Universal Robots PolyScope program: Bridge_big.urp

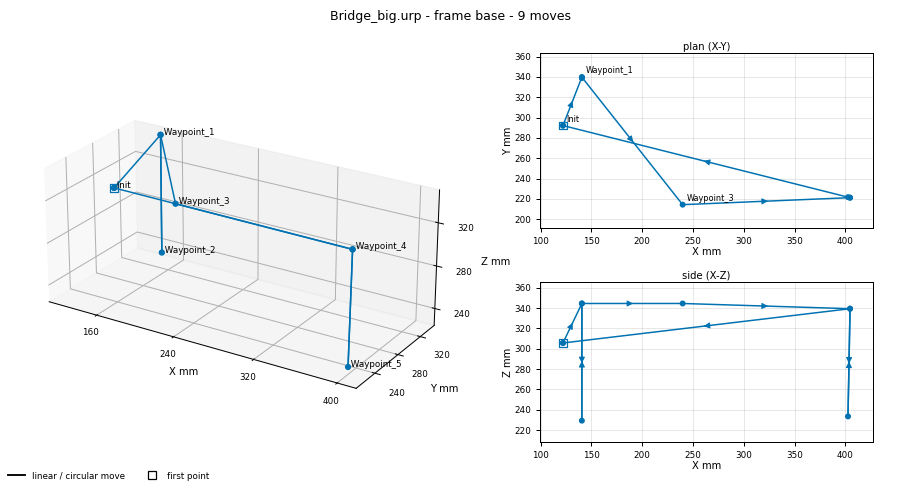
[picture p0: tool path of Bridge_big.urp in frame base, 9 of 9 moves have a stored position in this frame; points joined in program order, loops and branches not executed]
Program Bridge_big (installation=default directory=/programs/Mursal createdIn=5.11.11.1010533 lastSavedIn=5.11.11.1010533 robotSerialNumber=20205300864)
Calibrated DH parameters: a=[-0.000166, -0.243494, -0.153108, 0.000057, -0.000123, 0]; d=[0.151897, -1.34267, 53.988124, -52.514559, 0.085283, 0.092193]; alpha=[1.572472, -0.003756, 0.002824, 1.570807, -1.572621, 0]; deltaTheta=[0, 0.020704, 7.033215, -0.770746, 0.000004, 0]
Robot Program (runOnlyOnce=false)
  MoveL speed 250 mm/s, acceleration 1200 mm/s^2 (useActiveTCP=true) feature=Base
    Waypoint Init: TCP in base x=122.097 y=292.134 z=305.712 mm, rx=1.1347 ry=-2.9294 rz=0 rad; joints [91.644, -87.589, -91.768, -90.539, 90.036, 859.397] deg
    Waypoint Waypoint_1: TCP in base x=140.703 y=339.677 z=344.565 mm, rx=-2.2692 ry=2.1726 rz=0 rad; joints [88.306, -101.866, -65.574, -102.453, 89.953, 805.891] deg
    Waypoint Waypoint_2: TCP in base x=140.681 y=338.804 z=229.296 mm, rx=-2.2693 ry=2.1725 rz=0.0001 rad; joints [88.246, -103.09, -95.448, -71.353, 90.007, 805.889] deg
    URCap Gripper (Robotiq_Grippers, Robotiq Inc.) dataModel(position=100.0, force=100.0, speed=60.0, positionInDouble=100.0, forceInDouble=100.0, speedInDouble=60.0, slaveIds=[9], blocking=true, robotCompliant=false)
    Waypoint Waypoint_1: TCP in base x=140.703 y=339.677 z=344.565 mm, rx=-2.2692 ry=2.1726 rz=0 rad; joints [88.306, -101.866, -65.574, -102.453, 89.953, 805.891] deg
    Waypoint Waypoint_3: TCP in base x=239.819 y=214.305 z=344.563 mm, rx=-2.2692 ry=2.1726 rz=0.0001 rad; joints [65.729, -89.813, -79.085, -100.996, 90.004, 783.322] deg
    Waypoint Waypoint_4: TCP in base x=404.489 y=221.183 z=339.433 mm, rx=2.2692 ry=-2.1726 rz=-0.0001 rad; joints [45.209, -135.333, -14.024, -120.541, 89.8, 762.717] deg
    Waypoint Waypoint_5: TCP in base x=402.481 y=221.679 z=233.467 mm, rx=-2.2417 ry=2.2009 rz=0.0001 rad; joints [45.337, -125.997, -60.267, -83.629, 89.911, 764.361] deg
    URCap Gripper (Robotiq_Grippers, Robotiq Inc.) dataModel(position=0.0, force=0.7647058823529402, speed=100.0, positionInDouble=0.0, forceInDouble=0.7647058823529402, speedInDouble=100.0, slaveIds=[9], blocking=true, robotCompliant=false)
    Waypoint Waypoint_4: TCP in base x=404.489 y=221.183 z=339.433 mm, rx=2.2692 ry=-2.1726 rz=-0.0001 rad; joints [45.209, -135.333, -14.024, -120.541, 89.8, 762.717] deg
    Waypoint Init: TCP in base x=122.097 y=292.134 z=305.712 mm, rx=1.1347 ry=-2.9294 rz=0 rad; joints [91.644, -87.589, -91.768, -90.539, 90.036, 859.397] deg
